FUNCTION_BLOCK L3_PPTable (* Service Interface Function Block Type *)
  (* Standard: 61499-2 *)
  (* Version 0.0, 2014-11-06, EQUEROL, UJI *)
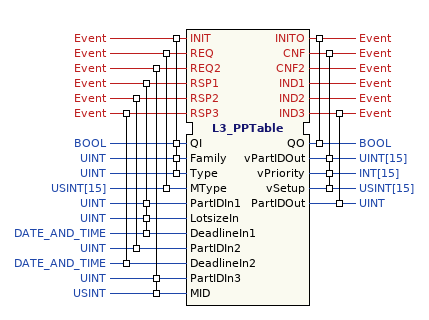
  EVENT_INPUT
    INIT WITH QI, Family, Type; (* Service Initialization *)
    REQ WITH MType; (* Service Request *)
    REQ2 WITH MID, PartIDIn3; (* Service request 2 *)
    RSP1 WITH PartIDIn1, LotsizeIn, DeadlineIn1; (* Application Response to IND *)
    RSP2 WITH PartIDIn2; (* Application Response to IND *)
    RSP3 WITH DeadlineIn2; (* Application Response to IND *)
  END_EVENT
  EVENT_OUTPUT
    INITO WITH QO; (* Initialization Confirm *)
    CNF WITH vPartIDOut, vPriority, vSetup; (* Confirmation of Requested Service *)
    CNF2; (* Request 2 execution confirm *)
    IND1; (* Indication from Resource *)
    IND2; (* Indication from Resource *)
    IND3 WITH PartIDOut; (* Indication from Resource *)
  END_EVENT
  VAR_INPUT
    QI : BOOL; (* Event Input Qualifier *)
    Family : UINT; (* Process plan family *)
    Type : UINT; (* Process plan type *)
    MType : ARRAY [0..14] OF USINT; (* Machine types vector *)
    PartIDIn1 : UINT; (* Part identifier *)
    LotsizeIn : UINT; (* Number of parts to be manufactured *)
    DeadlineIn1 : DATE_AND_TIME; (* Parts delivery time *)
    PartIDIn2 : UINT; (* Part identifier *)
    DeadlineIn2 : DATE_AND_TIME; (* Delivery time *)
    PartIDIn3 : UINT; (* Part identifier *)
    MID : USINT; (* Machine identifier *)
  END_VAR
  VAR_OUTPUT
    QO : BOOL; (* Event Output Qualifier *)
    vPartIDOut : ARRAY [0..14] OF UINT; (* Vector of parts used in the assignation *)
    vPriority : ARRAY [0..14] OF INT; (* Vector of priorities *)
    vSetup : ARRAY [0..14] OF USINT; (* Vector of setups *)
    PartIDOut : UINT; (* Part identifier *)
  END_VAR
  SERVICE APPLICATION/RESOURCE (* Service Interface Function Block Type *)
    SEQUENCE normal_establishment
      APPLICATION.INIT+(PARAMS) -> APPLICATION.INITO+(PARAMS);
    END_SEQUENCE
    SEQUENCE unsuccessful_establishment
      APPLICATION.INIT+(PARAMS) -> APPLICATION.INITO-(STATUS);
    END_SEQUENCE
    SEQUENCE request_confirm
      APPLICATION.REQ+(SD) -> APPLICATION.CNF+(RD);
    END_SEQUENCE
    SEQUENCE request_inhibited
      APPLICATION.REQ-(SD) -> APPLICATION.CNF-(STATUS);
    END_SEQUENCE
    SEQUENCE request_error
      APPLICATION.REQ+(SD) -> APPLICATION.CNF-(STATUS);
    END_SEQUENCE
    SEQUENCE indication_response
      RESOURCE.indicate(RD) -> APPLICATION.IND+(RD);
      APPLICATION.RSP(QI,SD) -> RESOURCE.response(QI,SD);
    END_SEQUENCE
    SEQUENCE indication_inhibited
      RESOURCE.indicate(RD,QI=FALSE) -> RESOURCE.inhibited();
    END_SEQUENCE
    SEQUENCE error_indication
      RESOURCE.error(STATUS) -> APPLICATION.IND-(STATUS);
    END_SEQUENCE
    SEQUENCE application_initiated_termination
      APPLICATION.INIT-() -> APPLICATION.INITO-(STATUS);
    END_SEQUENCE
    SEQUENCE resource_initiated_termination
      -> APPLICATION.INITO-(STATUS);
    END_SEQUENCE
  END_SERVICE
END_FUNCTION_BLOCK
